TYPE ST_GC_ServiceStatus :
STRUCT
	SpinAxisJog : ST_GCSpinAxisJogStatus;
	SpinAxisMoveAbs : ST_GCSpinAxisMoveAbsStatus;
END_STRUCT
END_TYPE

(* stored: Version 1.1.0.1, ProductVersion 3.1.4026.18
   DUT ST_GC_ServiceStatus: Id {f27be8ff-16cd-4df7-a4df-6e0527b043a3} *)
